Staubli VAL3: clkStop.pgx

program clkStop()
begin
  bDoAirex = false
  bDoModules = false
  bCleanup = false
end
